TYPE ST_BatterySections EXTENDS ST_SectionBase :
STRUCT
END_STRUCT
END_TYPE

(* stored: Version 1.1.0.1, ProductVersion 3.1.4024.12
   DUT ST_BatterySections: Id {ae92fb29-7195-4c1b-9a04-82e42d4106c5} *)
